Fanuc KAREL source: kt00005.KL

-- PROVISIONAL review KL for V940-1; original PC SHA256 097d6fb57a654c5fc6a8f5f6945c6b97954c810fef39d96600761de13d583104
-- Incomplete behavior may be omitted. Consult companion uncertainty JSON. Do not deploy.
PROGRAM KT00005
%NOLOCKGROUP
VAR
  I1 : INTEGER
  OUT : INTEGER
-- UNRESOLVED_DECL Y2 type=002018
BEGIN
  -- V9_ZERO_TABLE_METADATA_HINT layout=0001; no indexed target words; source/name/runtime held
  -- UNRESOLVED_PC offsets 5-16; opcodes 2E,23
  -- UNRESOLVED_PC offsets 21-35; opcodes 2E,22,9D,33,B2
  -- UNRESOLVED_PC offsets 40-62; opcodes 21,22,9D,33,B1,52,23
  -- UNRESOLVED_PC offsets 67-71; opcodes 7F
END KT00005
